FUNCTION_BLOCK fbRealToWord
VAR_INPUT
	in_r_Value				: REAL ;
	in_r_Res				: REAL ;
	in_i_Offset				: INT ;
END_VAR
VAR_OUTPUT
	out_B0					: BYTE ;
	out_B1					: BYTE ;
END_VAR
VAR
	w_AddedValue			: WORD;
	r_ResolutionResolved	: REAL;
	r_OffsetSolved			: REAL;
END_VAR

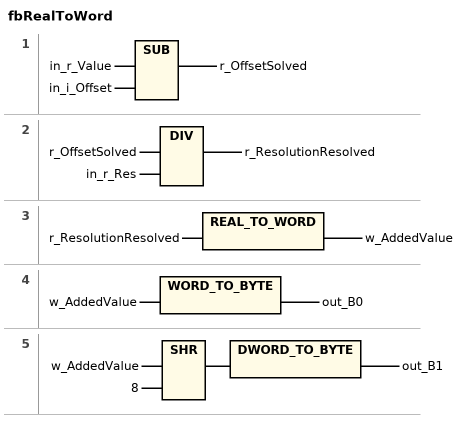
// NETWORK 1
r_OffsetSolved := in_r_Value - in_i_Offset;

// NETWORK 2
r_ResolutionResolved := r_OffsetSolved / in_r_Res;

// NETWORK 3
w_AddedValue := REAL_TO_WORD(r_ResolutionResolved);

// NETWORK 4
out_B0 := WORD_TO_BYTE(w_AddedValue);

// NETWORK 5
out_B1 := DWORD_TO_BYTE(SHR(w_AddedValue, 8));

END_FUNCTION_BLOCK

(* stored: Version 1.1.0.1, ProductVersion 3.1.4024.12
   POU fbRealToWord: Id {28cf3834-f931-48af-b535-6682a285d5bf}, SpecialFunc None *)
